INTERFACE ITF_ModuleSequenceControl

METHOD ClearSequence : BOOL
VAR_INPUT
END_VAR
END_METHOD

METHOD DisableSequence : BOOL
END_METHOD

METHOD EnableSequence : BOOL
END_METHOD

METHOD ResetSequence : BOOL
END_METHOD

METHOD ResumeSequence : BOOL
VAR_INPUT
END_VAR
END_METHOD

PROPERTY SequenceCommand : E_ModuleSequenceCommand
GET
END_GET
SET
END_SET
END_PROPERTY

PROPERTY SequenceStatus : E_ModuleSequenceStatus
GET
END_GET
END_PROPERTY

METHOD StartSequence : BOOL
END_METHOD

END_INTERFACE

(* stored: Version 1.1.0.1, ProductVersion 3.1.4024.9
   Itf ITF_ModuleSequenceControl: Id {52a4eb92-e318-455a-b036-1d096da524a0}
   Folder 01_Properties: Id {32cd75db-95e6-4e59-a337-d34f54cfaff6}
   Folder 02_Methods: Id {f5543132-710e-4d85-a828-6df720f8cd24}
   Method ClearSequence: Id {056019a7-2e4c-42d1-a163-e1caa0b45df2}
   Method DisableSequence: Id {065e23ff-b747-413c-8d73-70bd3d6bf772}
   Method EnableSequence: Id {f50796c5-0747-4cbf-a675-cfdcbdde6337}
   Method ResetSequence: Id {e7ff7a2f-11b6-4f0a-8c69-bc4d4a42a02b}
   Method ResumeSequence: Id {f5b31e9a-e3be-450c-8d6c-d87e7c3eaab5}
   Property SequenceCommand: Id {0ebfd7d8-a88a-4f68-9367-23775a846165}
   Get Get: Id {46bb49a3-6de1-4514-a212-ce92f23e5a5a}
   Set Set: Id {f5e82b1e-12e3-49bc-a15a-e9bab737f18f}
   Property SequenceStatus: Id {dc623bca-b670-4005-9e61-b94aedaaf083}
   Get Get: Id {49621555-2b99-4be8-9a88-35bb80aaeb73}
   Method StartSequence: Id {b110fc19-185b-4e21-93ff-0aef69c44f70} *)
